INTERFACE I_Observer EXTENDS __SYSTEM.IQueryInterface, I_Equatable

METHOD OnError
VAR_INPUT
END_VAR
END_METHOD

METHOD OnUpdate
VAR_INPUT
END_VAR
END_METHOD

END_INTERFACE

(* stored: Version 1.1.0.1, ProductVersion 3.1.4024.6
   Itf I_Observer: Id {124708d7-5f22-4283-b4ac-818df7ab3030}
   Method OnError: Id {b8c25812-ba2f-4a94-a971-ce9519865e34}
   Method OnUpdate: Id {8d2f5007-6386-470c-aa20-0f3022466b5d} *)
